(* Logix 5000 project; controller STAT 1756-L72 rev 20.12; software revision 20.04; part 19 of 34 *)
(* tags used below, declared in another part *)
   B14 : DINT[30];
   B16 : DINT[30];
   B17 : DINT[30];
   B3 : DINT[256];
   B9 : DINT[40];
   F8 : REAL[256];
   I1_005_Bit15 : ALIAS FOR I1[5].15;
   I6_000_Bit02 : ALIAS FOR I6[0].2;   // totaal 3 debiet stfa 3
   I6_000_Bit10 : ALIAS FOR I6[0].10;   // pressostaat osmose1
   I6_000_Bit11 : ALIAS FOR I6[0].11;   // pressostaat osmose2
   I6_000_Bit12 : ALIAS FOR I6[0].12;   // pressostaat osmose3
   I6_001_Bit07 : ALIAS FOR I6[1].7;   // pulse debietmeter zandfilter osmose
   N12 : DINT[230];
   N13 : DINT[230];
   N26 : DINT[256];
   O14_000_Bit14 : ALIAS FOR O14[0].14;   // STFA3_EV1 STFA3_EV1
   O14_000_Bit15 : ALIAS FOR O14[0].15;   // STFA3_EV2 STFA3_EV2
   O14_001_Bit00 : ALIAS FOR O14[1].0;   // STFA3_EV3 STFA3_EV3
   O14_001_Bit01 : ALIAS FOR O14[1].1;   // STFA3_EV4 STFA3_EV4
   O14_001_Bit02 : ALIAS FOR O14[1].2;   // STFA3_EV5 STFA3_EV5
   O14_001_Bit03 : ALIAS FOR O14[1].3;   // STFA3_EV6 STFA3_EV6
   O14_001_Bit12 : ALIAS FOR O14[1].12;   // RO1_EV1 RO1_EV1
   O14_001_Bit13 : ALIAS FOR O14[1].13;   // RO1_EV2 RO1_EV2
   O15_000_Bit00 : ALIAS FOR O15[0].0;   // RO2_EV1 RO2_EV1
   O15_000_Bit01 : ALIAS FOR O15[0].1;   // RO2_EV2 RO2_EV2
   T27 : TIMER[100];
   T4 : TIMER[200];
(* ibt, continued *)

ROUTINE _22_SEQ_VERZ3   (* ladder *)
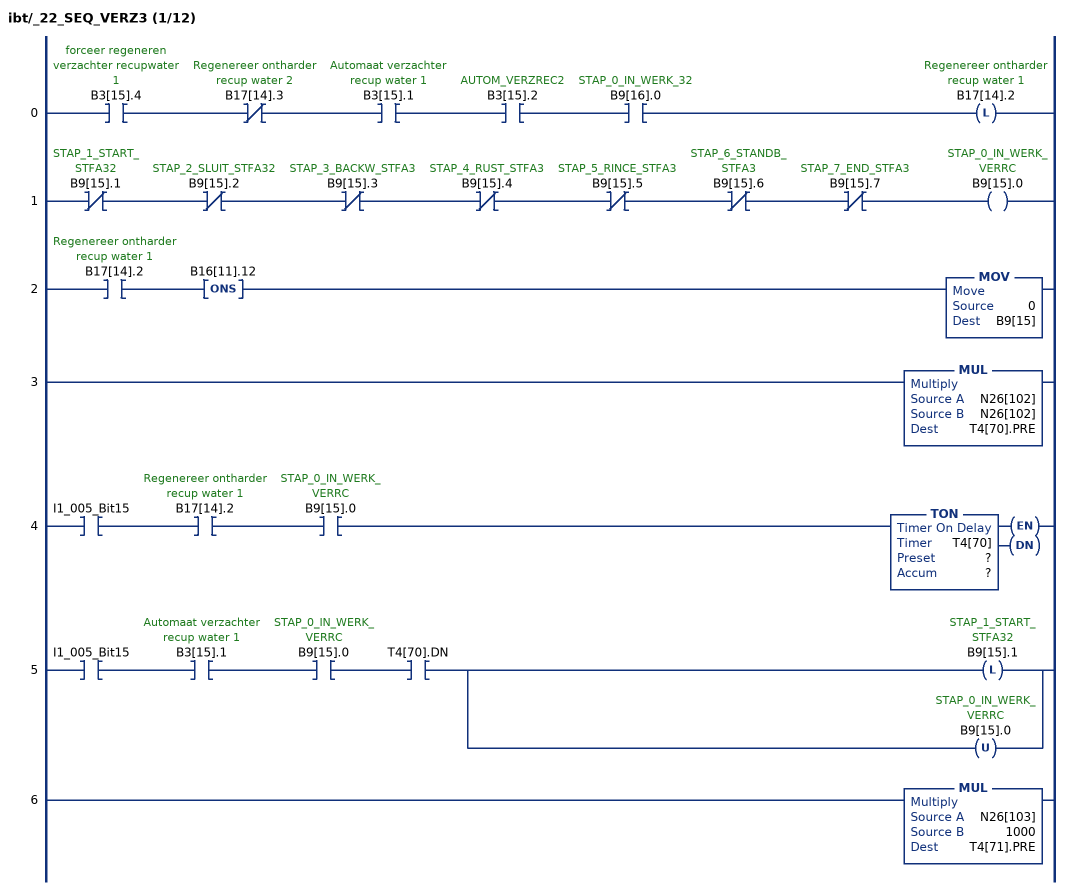
   0: XIC(B3[15].4)XIO(B17[14].3)XIC(B3[15].1)XIC(B3[15].2)XIC(B9[16].0)OTL(B17[14].2);
   1: XIO(B9[15].1)XIO(B9[15].2)XIO(B9[15].3)XIO(B9[15].4)XIO(B9[15].5)XIO(B9[15].6)XIO(B9[15].7)OTE(B9[15].0);
   2: XIC(B17[14].2)ONS(B16[11].12)MOV(0,B9[15]);
   3: MUL(N26[102],N26[102],T4[70].PRE);
   4: XIC(I1_005_Bit15)XIC(B17[14].2)XIC(B9[15].0)TON(T4[70],?,?);
   5: XIC(I1_005_Bit15)XIC(B3[15].1)XIC(B9[15].0)XIC(T4[70].DN)[OTL(B9[15].1) ,OTU(B9[15].0) ];
   6: MUL(N26[103],1000,T4[71].PRE);
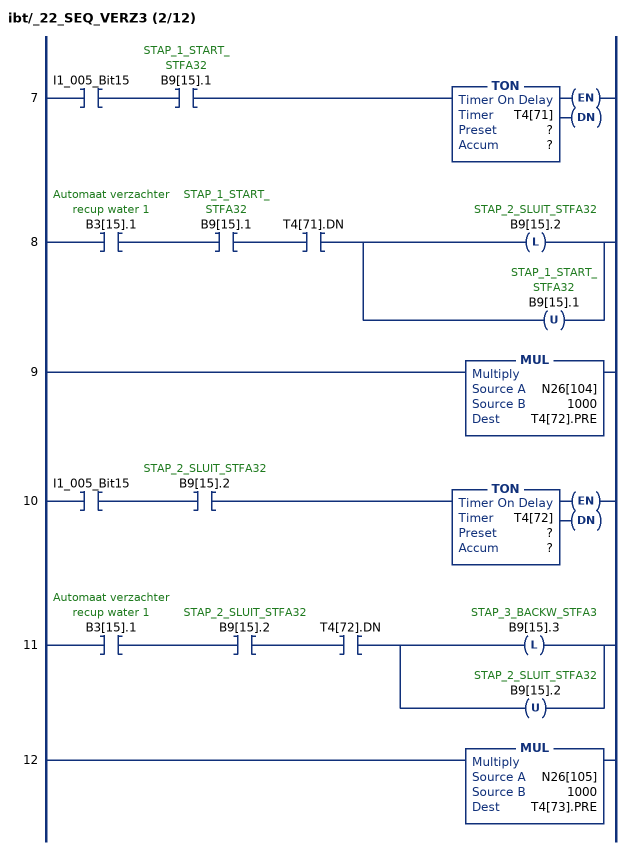
   7: XIC(I1_005_Bit15)XIC(B9[15].1)TON(T4[71],?,?);
   8: XIC(B3[15].1)XIC(B9[15].1)XIC(T4[71].DN)[OTL(B9[15].2) ,OTU(B9[15].1) ];
   9: MUL(N26[104],1000,T4[72].PRE);
   10: XIC(I1_005_Bit15)XIC(B9[15].2)TON(T4[72],?,?);
   11: XIC(B3[15].1)XIC(B9[15].2)XIC(T4[72].DN)[OTL(B9[15].3) ,OTU(B9[15].2) ];
   12: MUL(N26[105],1000,T4[73].PRE);
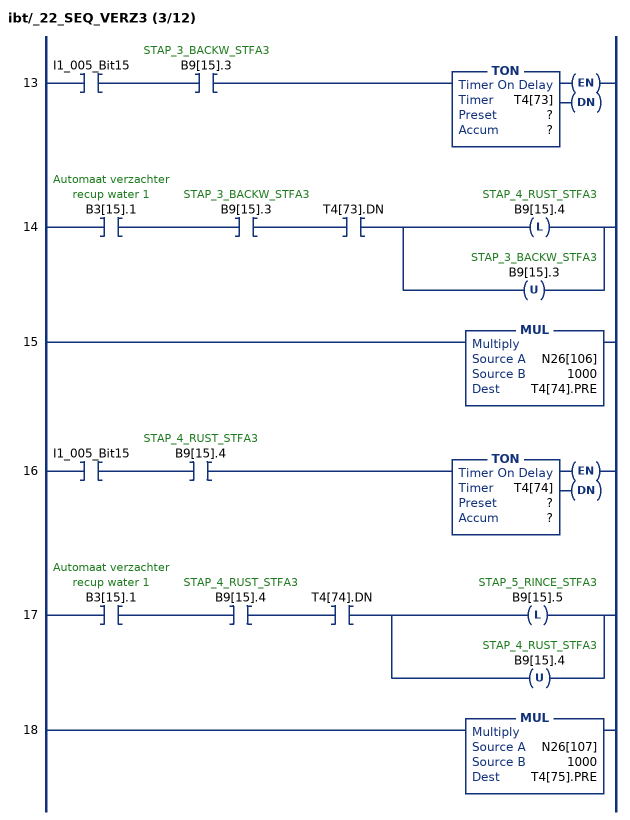
   13: XIC(I1_005_Bit15)XIC(B9[15].3)TON(T4[73],?,?);
   14: XIC(B3[15].1)XIC(B9[15].3)XIC(T4[73].DN)[OTL(B9[15].4) ,OTU(B9[15].3) ];
   15: MUL(N26[106],1000,T4[74].PRE);
   16: XIC(I1_005_Bit15)XIC(B9[15].4)TON(T4[74],?,?);
   17: XIC(B3[15].1)XIC(B9[15].4)XIC(T4[74].DN)[OTL(B9[15].5) ,OTU(B9[15].4) ];
   18: MUL(N26[107],1000,T4[75].PRE);
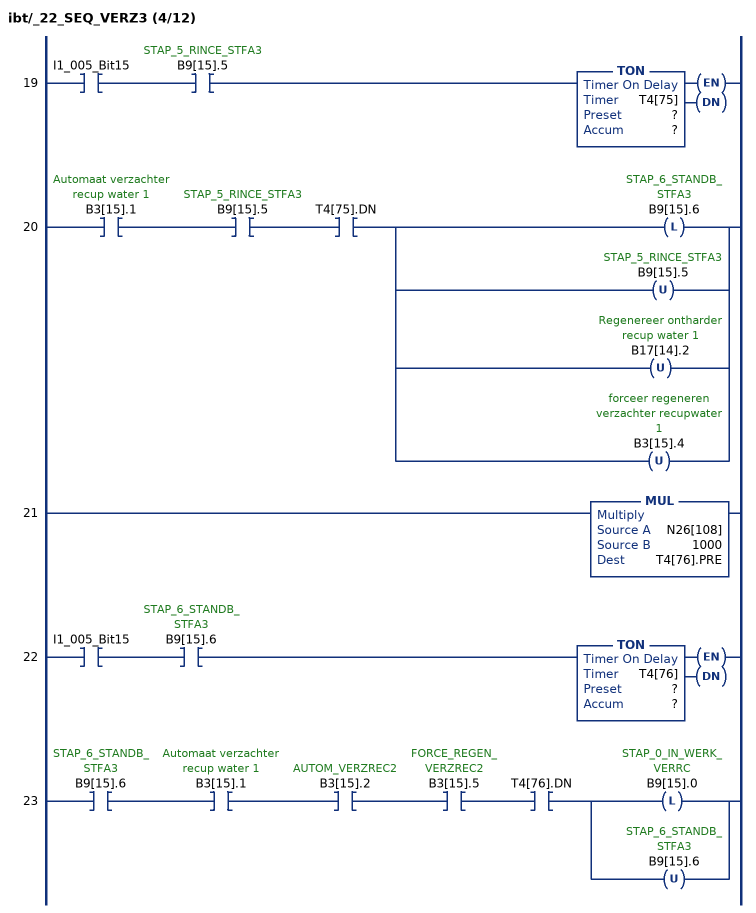
   19: XIC(I1_005_Bit15)XIC(B9[15].5)TON(T4[75],?,?);
   20: XIC(B3[15].1)XIC(B9[15].5)XIC(T4[75].DN)[OTL(B9[15].6) ,[OTU(B9[15].5) ,[OTU(B17[14].2) ,OTU(B3[15].4) ] ] ];
   21: MUL(N26[108],1000,T4[76].PRE);
   22: XIC(I1_005_Bit15)XIC(B9[15].6)TON(T4[76],?,?);
   23: XIC(B9[15].6)XIC(B3[15].1)XIC(B3[15].2)XIC(B3[15].5)XIC(T4[76].DN)[OTL(B9[15].0) ,OTU(B9[15].6) ];
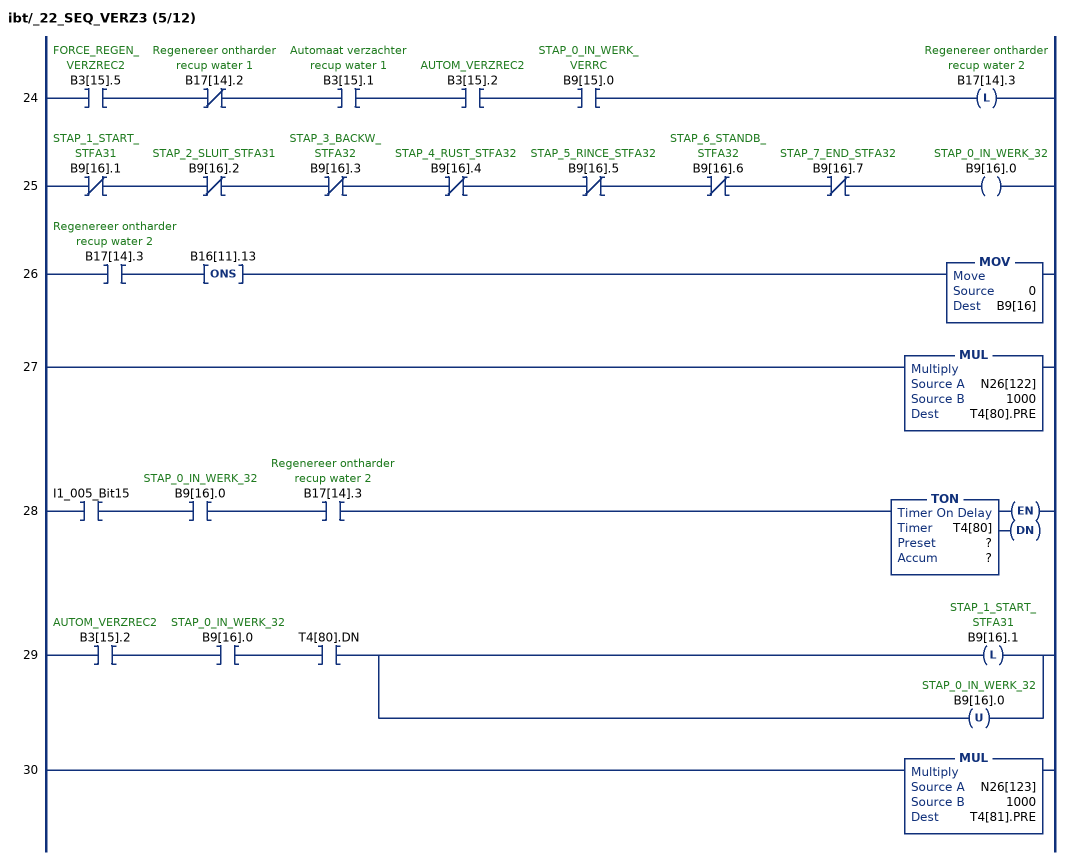
   24: XIC(B3[15].5)XIO(B17[14].2)XIC(B3[15].1)XIC(B3[15].2)XIC(B9[15].0)OTL(B17[14].3);
   25: XIO(B9[16].1)XIO(B9[16].2)XIO(B9[16].3)XIO(B9[16].4)XIO(B9[16].5)XIO(B9[16].6)XIO(B9[16].7)OTE(B9[16].0);
   26: XIC(B17[14].3)ONS(B16[11].13)MOV(0,B9[16]);
   27: MUL(N26[122],1000,T4[80].PRE);
   28: XIC(I1_005_Bit15)XIC(B9[16].0)XIC(B17[14].3)TON(T4[80],?,?);
   29: XIC(B3[15].2)XIC(B9[16].0)XIC(T4[80].DN)[OTL(B9[16].1) ,OTU(B9[16].0) ];
   30: MUL(N26[123],1000,T4[81].PRE);
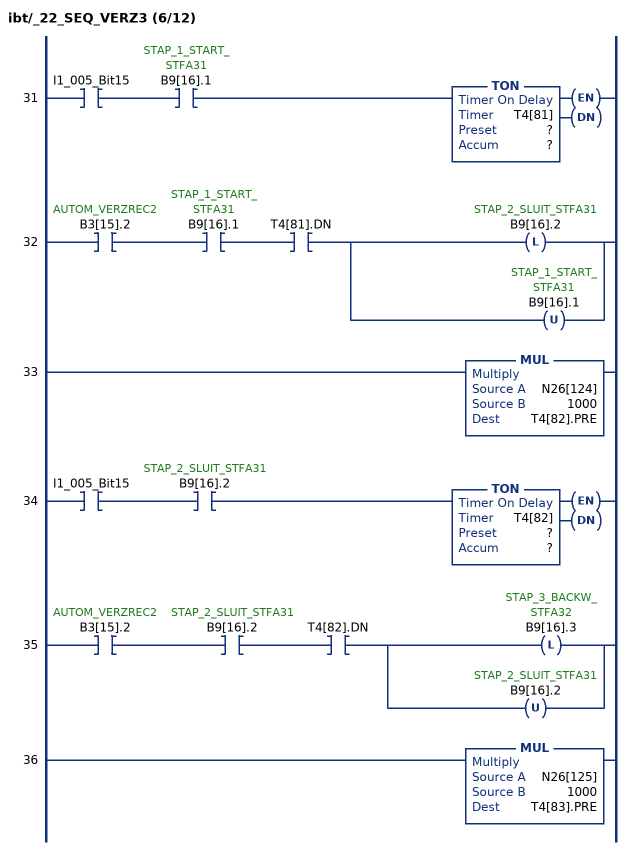
   31: XIC(I1_005_Bit15)XIC(B9[16].1)TON(T4[81],?,?);
   32: XIC(B3[15].2)XIC(B9[16].1)XIC(T4[81].DN)[OTL(B9[16].2) ,OTU(B9[16].1) ];
   33: MUL(N26[124],1000,T4[82].PRE);
   34: XIC(I1_005_Bit15)XIC(B9[16].2)TON(T4[82],?,?);
   35: XIC(B3[15].2)XIC(B9[16].2)XIC(T4[82].DN)[OTL(B9[16].3) ,OTU(B9[16].2) ];
   36: MUL(N26[125],1000,T4[83].PRE);
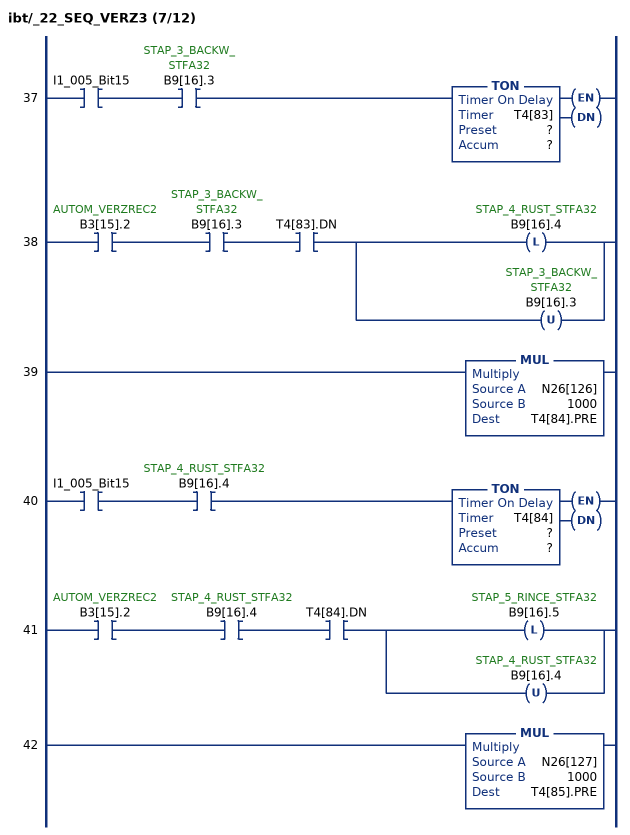
   37: XIC(I1_005_Bit15)XIC(B9[16].3)TON(T4[83],?,?);
   38: XIC(B3[15].2)XIC(B9[16].3)XIC(T4[83].DN)[OTL(B9[16].4) ,OTU(B9[16].3) ];
   39: MUL(N26[126],1000,T4[84].PRE);
   40: XIC(I1_005_Bit15)XIC(B9[16].4)TON(T4[84],?,?);
   41: XIC(B3[15].2)XIC(B9[16].4)XIC(T4[84].DN)[OTL(B9[16].5) ,OTU(B9[16].4) ];
   42: MUL(N26[127],1000,T4[85].PRE);
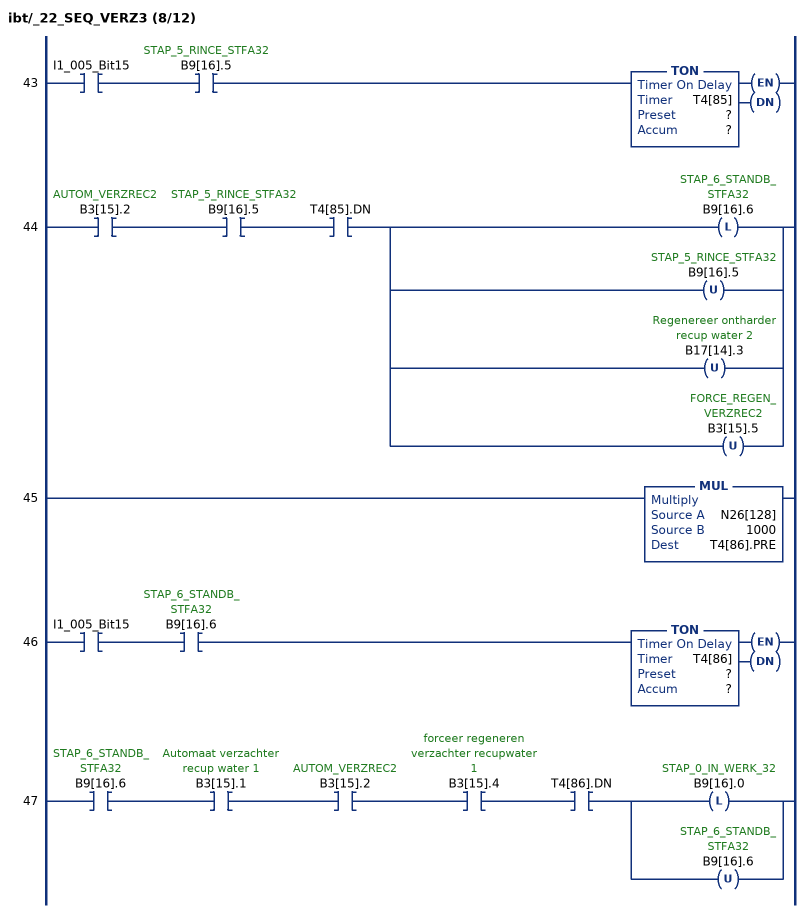
   43: XIC(I1_005_Bit15)XIC(B9[16].5)TON(T4[85],?,?);
   44: XIC(B3[15].2)XIC(B9[16].5)XIC(T4[85].DN)[OTL(B9[16].6) ,[OTU(B9[16].5) ,[OTU(B17[14].3) ,OTU(B3[15].5) ] ] ];
   45: MUL(N26[128],1000,T4[86].PRE);
   46: XIC(I1_005_Bit15)XIC(B9[16].6)TON(T4[86],?,?);
   47: XIC(B9[16].6)XIC(B3[15].1)XIC(B3[15].2)XIC(B3[15].4)XIC(T4[86].DN)[OTL(B9[16].0) ,OTU(B9[16].6) ];
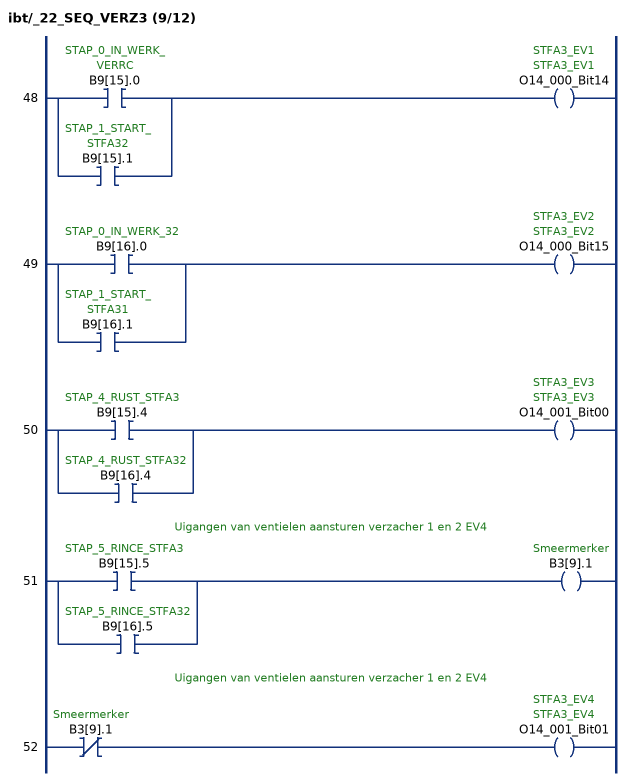
   48: [XIC(B9[15].0) ,XIC(B9[15].1) ]OTE(O14_000_Bit14);
   49: [XIC(B9[16].0) ,XIC(B9[16].1) ]OTE(O14_000_Bit15);
   50: [XIC(B9[15].4) ,XIC(B9[16].4) ]OTE(O14_001_Bit00);
   // Uigangen van ventielen aansturen verzacher 1 en 2 EV4
   51: [XIC(B9[15].5) ,XIC(B9[16].5) ]OTE(B3[9].1);
   // Uigangen van ventielen aansturen verzacher 1 en 2 EV4
   52: XIO(B3[9].1)OTE(O14_001_Bit01);
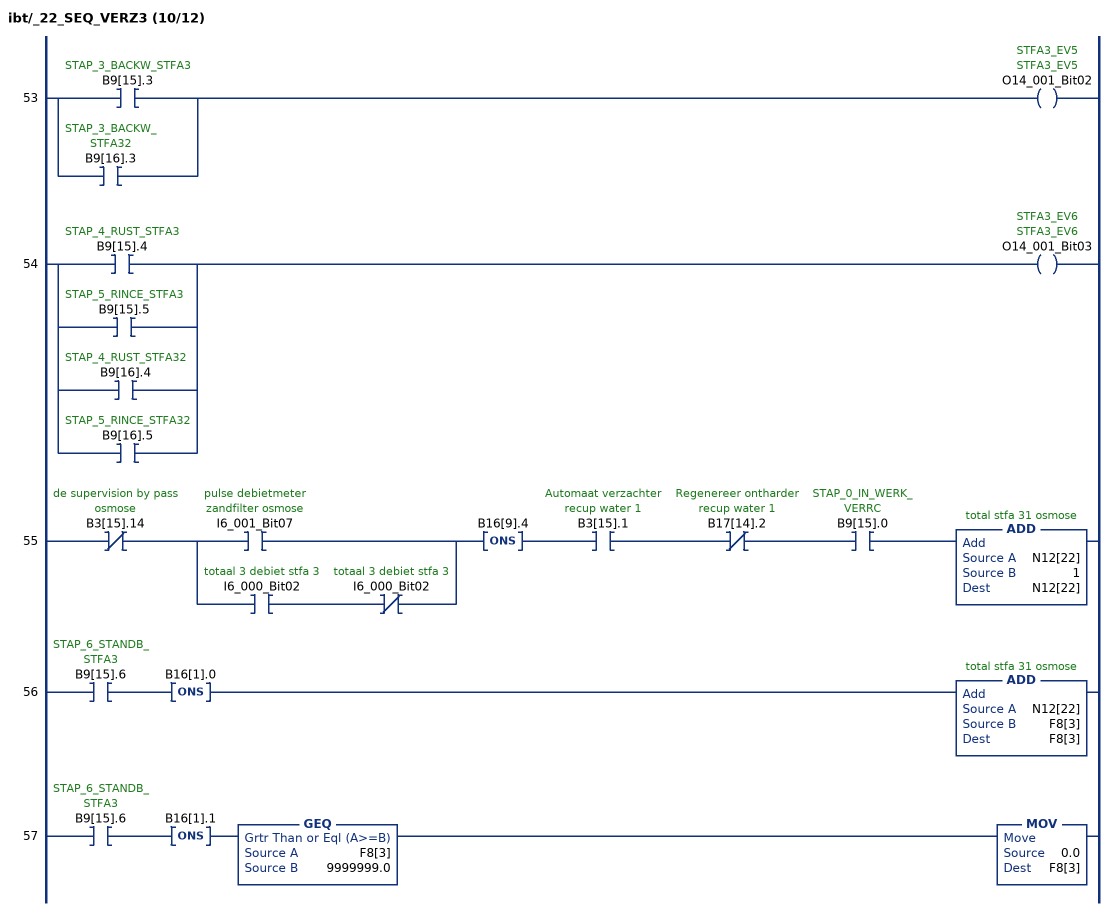
   53: [XIC(B9[15].3) ,XIC(B9[16].3) ]OTE(O14_001_Bit02);
   54: [XIC(B9[15].4) ,[XIC(B9[15].5) ,[XIC(B9[16].4) ,XIC(B9[16].5) ] ] ]OTE(O14_001_Bit03);
   55: XIO(B3[15].14)[XIC(I6_001_Bit07) ,XIC(I6_000_Bit02) XIO(I6_000_Bit02) ]ONS(B16[9].4)XIC(B3[15].1)XIO(B17[14].2)XIC(B9[15].0)ADD(N12[22],1,N12[22]);
   56: XIC(B9[15].6)ONS(B16[1].0)ADD(N12[22],F8[3],F8[3]);
   57: XIC(B9[15].6)ONS(B16[1].1)GEQ(F8[3],9999999.0)MOV(0.0,F8[3]);
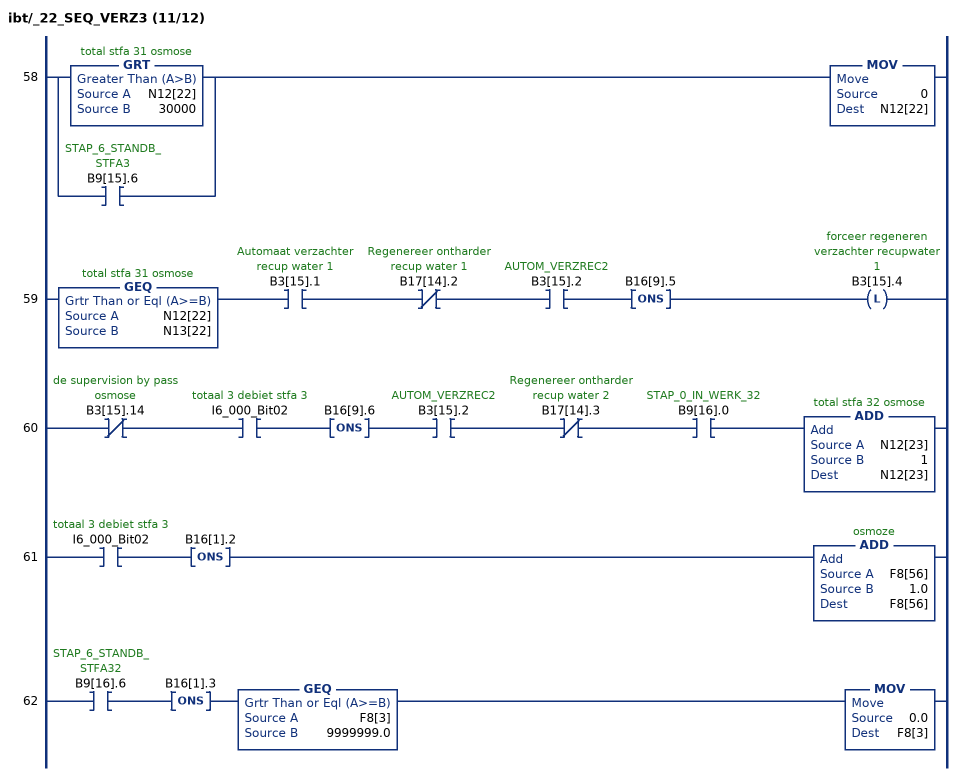
   58: [GRT(N12[22],30000) ,XIC(B9[15].6) ]MOV(0,N12[22]);
   59: GEQ(N12[22],N13[22])XIC(B3[15].1)XIO(B17[14].2)XIC(B3[15].2)ONS(B16[9].5)OTL(B3[15].4);
   60: XIO(B3[15].14)XIC(I6_000_Bit02)ONS(B16[9].6)XIC(B3[15].2)XIO(B17[14].3)XIC(B9[16].0)ADD(N12[23],1,N12[23]);
   61: XIC(I6_000_Bit02)ONS(B16[1].2)ADD(F8[56],1.0,F8[56]);
   62: XIC(B9[16].6)ONS(B16[1].3)GEQ(F8[3],9999999.0)MOV(0.0,F8[3]);
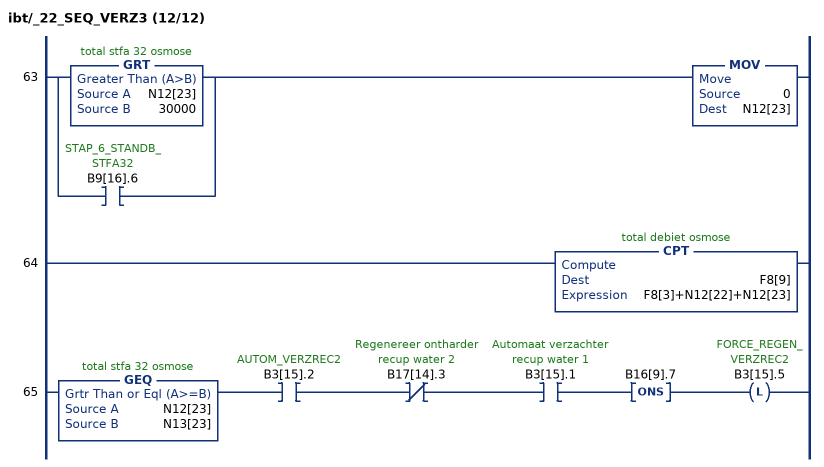
   63: [GRT(N12[23],30000) ,XIC(B9[16].6) ]MOV(0,N12[23]);
   64: CPT(F8[9],F8[3]+N12[22]+N12[23]);
   65: GEQ(N12[23],N13[23])XIC(B3[15].2)XIO(B17[14].3)XIC(B3[15].1)ONS(B16[9].7)OTL(B3[15].5);
END_ROUTINE

ROUTINE _23_SEQ_OSMOSE   (* ladder *)
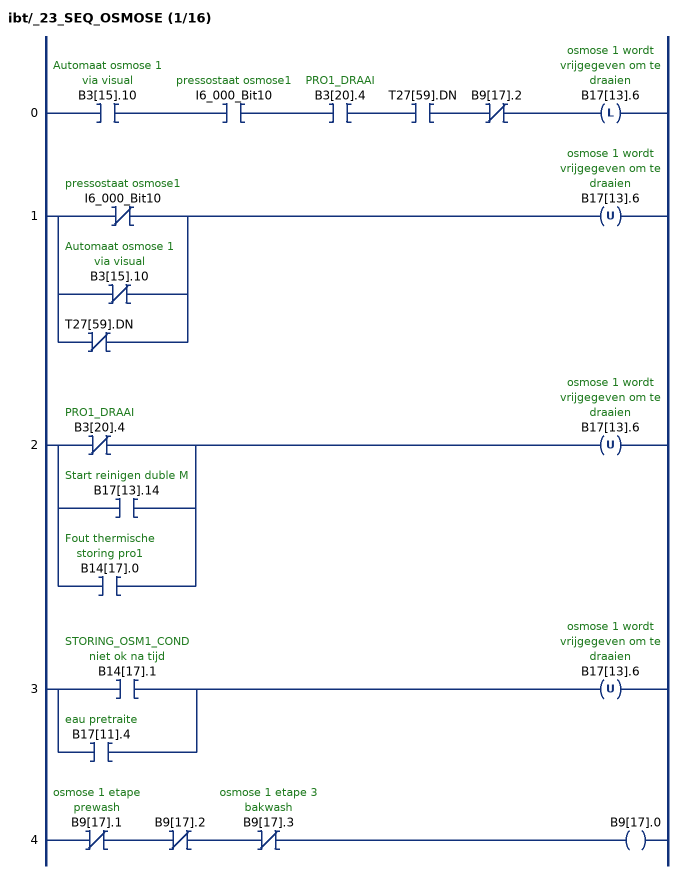
   0: XIC(B3[15].10)XIC(I6_000_Bit10)XIC(B3[20].4)XIC(T27[59].DN)XIO(B9[17].2)OTL(B17[13].6);
   1: [XIO(I6_000_Bit10) ,[XIO(B3[15].10) ,XIO(T27[59].DN) ] ]OTU(B17[13].6);
   2: [XIO(B3[20].4) ,[XIC(B17[13].14) ,XIC(B14[17].0) ] ]OTU(B17[13].6);
   3: [XIC(B14[17].1) ,XIC(B17[11].4) ]OTU(B17[13].6);
   4: XIO(B9[17].1)XIO(B9[17].2)XIO(B9[17].3)OTE(B9[17].0);
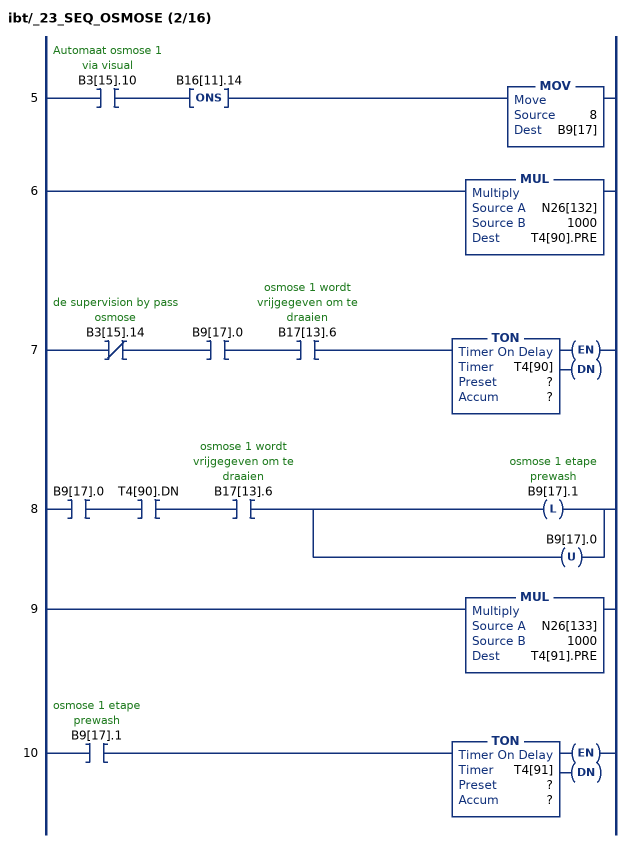
   5: XIC(B3[15].10)ONS(B16[11].14)MOV(8,B9[17]);
   6: MUL(N26[132],1000,T4[90].PRE);
   7: XIO(B3[15].14)XIC(B9[17].0)XIC(B17[13].6)TON(T4[90],?,?);
   8: XIC(B9[17].0)XIC(T4[90].DN)XIC(B17[13].6)[OTL(B9[17].1) ,OTU(B9[17].0) ];
   9: MUL(N26[133],1000,T4[91].PRE);
   10: XIC(B9[17].1)TON(T4[91],?,?);
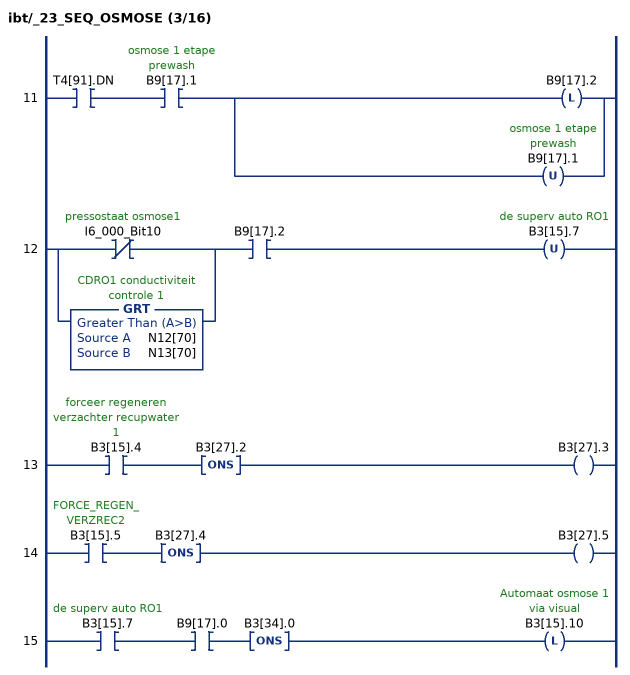
   11: XIC(T4[91].DN)XIC(B9[17].1)[OTL(B9[17].2) ,OTU(B9[17].1) ];
   12: [XIO(I6_000_Bit10) ,GRT(N12[70],N13[70]) ]XIC(B9[17].2)OTU(B3[15].7);
   13: XIC(B3[15].4)ONS(B3[27].2)OTE(B3[27].3);
   14: XIC(B3[15].5)ONS(B3[27].4)OTE(B3[27].5);
   15: XIC(B3[15].7)XIC(B9[17].0)ONS(B3[34].0)OTL(B3[15].10);
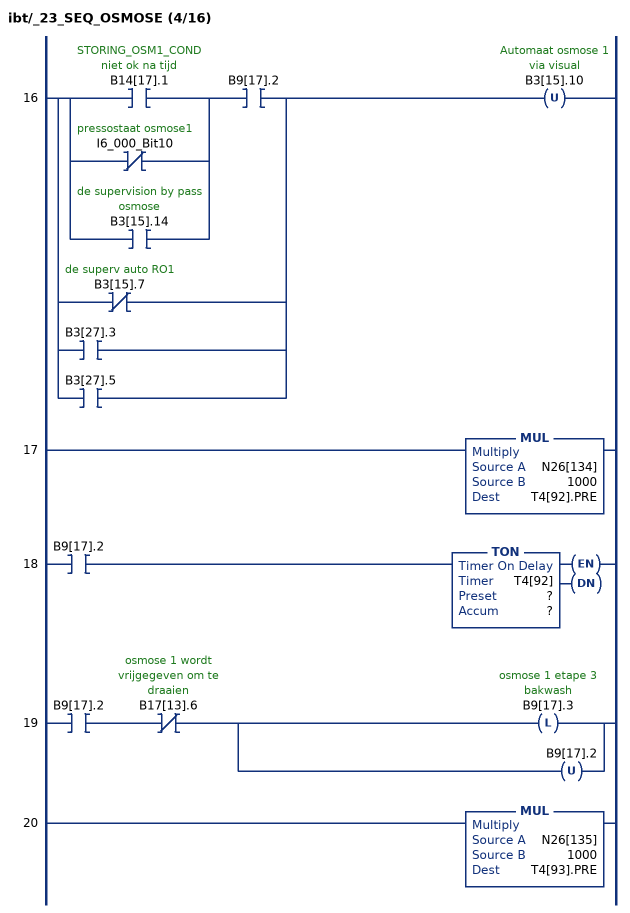
   16: [[XIC(B14[17].1) ,[XIO(I6_000_Bit10) ,XIC(B3[15].14) ] ] XIC(B9[17].2) ,XIO(B3[15].7) ,XIC(B3[27].3) ,XIC(B3[27].5) ]OTU(B3[15].10);
   17: MUL(N26[134],1000,T4[92].PRE);
   18: XIC(B9[17].2)TON(T4[92],?,?);
   19: XIC(B9[17].2)XIO(B17[13].6)[OTL(B9[17].3) ,OTU(B9[17].2) ];
   20: MUL(N26[135],1000,T4[93].PRE);
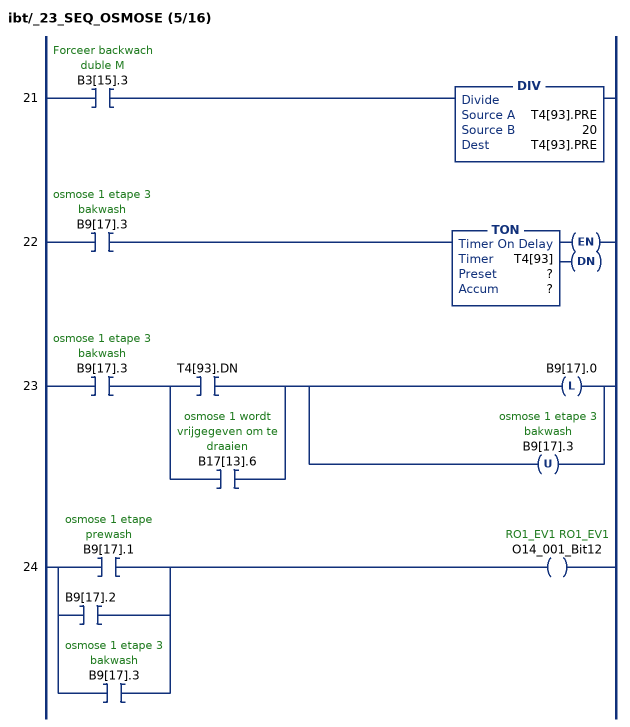
   21: XIC(B3[15].3)DIV(T4[93].PRE,20,T4[93].PRE);
   22: XIC(B9[17].3)TON(T4[93],?,?);
   23: XIC(B9[17].3)[XIC(T4[93].DN) ,XIC(B17[13].6) ][OTL(B9[17].0) ,OTU(B9[17].3) ];
   24: [XIC(B9[17].1) ,[XIC(B9[17].2) ,XIC(B9[17].3) ] ]OTE(O14_001_Bit12);
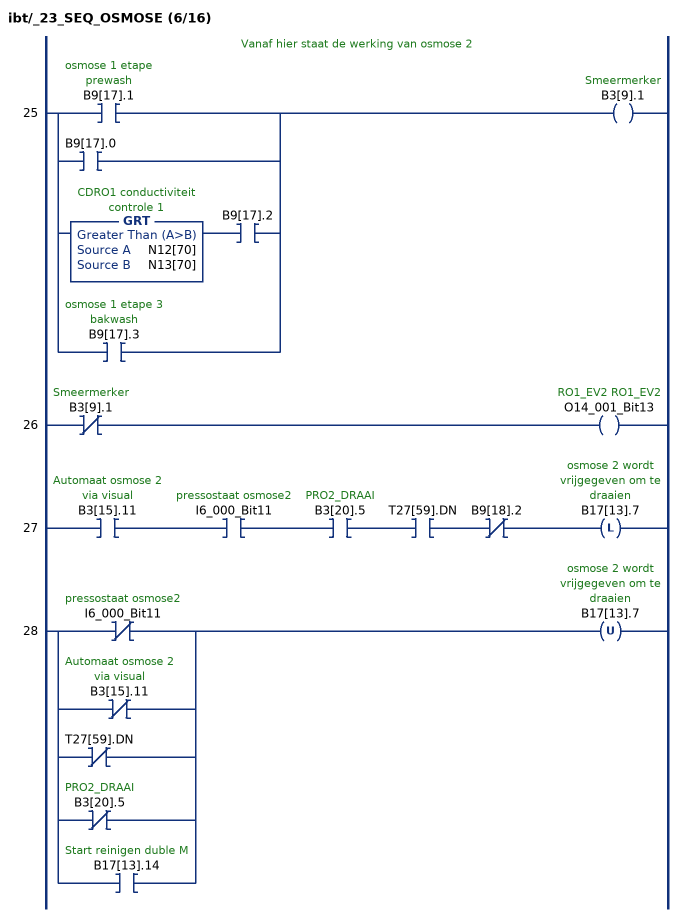
   // Vanaf hier staat de werking van osmose 2
   25: [[XIC(B9[17].1) ,XIC(B9[17].0) ] ,[GRT(N12[70],N13[70]) XIC(B9[17].2) ,XIC(B9[17].3) ] ]OTE(B3[9].1);
   26: XIO(B3[9].1)OTE(O14_001_Bit13);
   27: XIC(B3[15].11)XIC(I6_000_Bit11)XIC(B3[20].5)XIC(T27[59].DN)XIO(B9[18].2)OTL(B17[13].7);
   28: [XIO(I6_000_Bit11) ,[XIO(B3[15].11) ,[[XIO(T27[59].DN) ,XIO(B3[20].5) ] ,XIC(B17[13].14) ] ] ]OTU(B17[13].7);
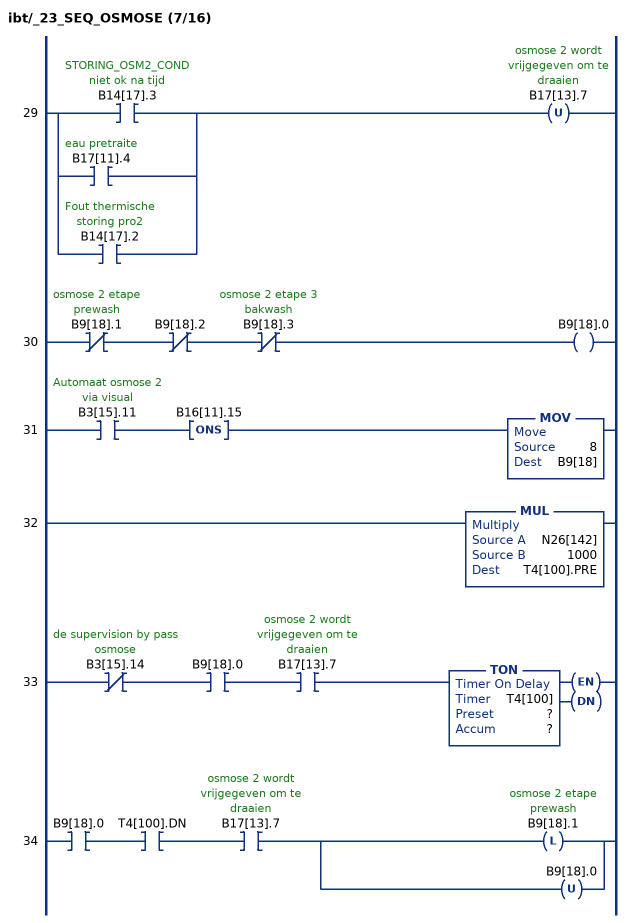
   29: [XIC(B14[17].3) ,[XIC(B17[11].4) ,XIC(B14[17].2) ] ]OTU(B17[13].7);
   30: XIO(B9[18].1)XIO(B9[18].2)XIO(B9[18].3)OTE(B9[18].0);
   31: XIC(B3[15].11)ONS(B16[11].15)MOV(8,B9[18]);
   32: MUL(N26[142],1000,T4[100].PRE);
   33: XIO(B3[15].14)XIC(B9[18].0)XIC(B17[13].7)TON(T4[100],?,?);
   34: XIC(B9[18].0)XIC(T4[100].DN)XIC(B17[13].7)[OTL(B9[18].1) ,OTU(B9[18].0) ];
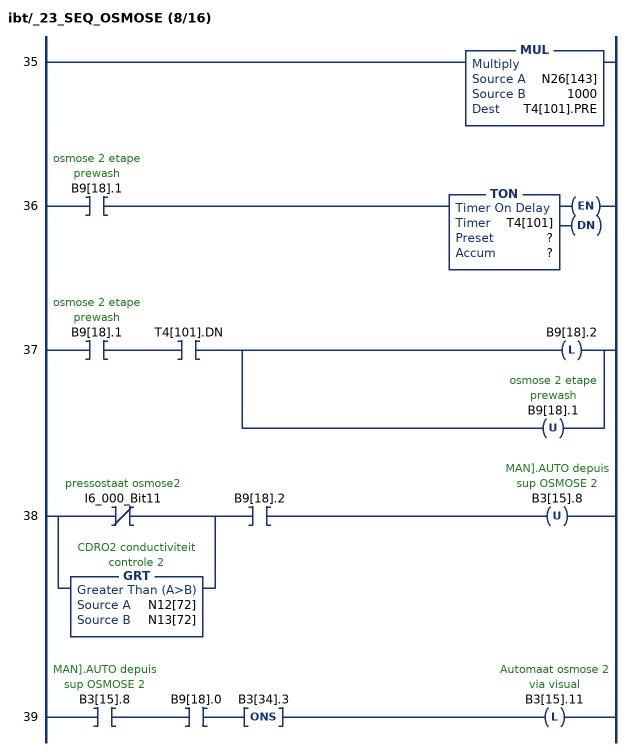
   35: MUL(N26[143],1000,T4[101].PRE);
   36: XIC(B9[18].1)TON(T4[101],?,?);
   37: XIC(B9[18].1)XIC(T4[101].DN)[OTL(B9[18].2) ,OTU(B9[18].1) ];
   38: [XIO(I6_000_Bit11) ,GRT(N12[72],N13[72]) ]XIC(B9[18].2)OTU(B3[15].8);
   39: XIC(B3[15].8)XIC(B9[18].0)ONS(B3[34].3)OTL(B3[15].11);
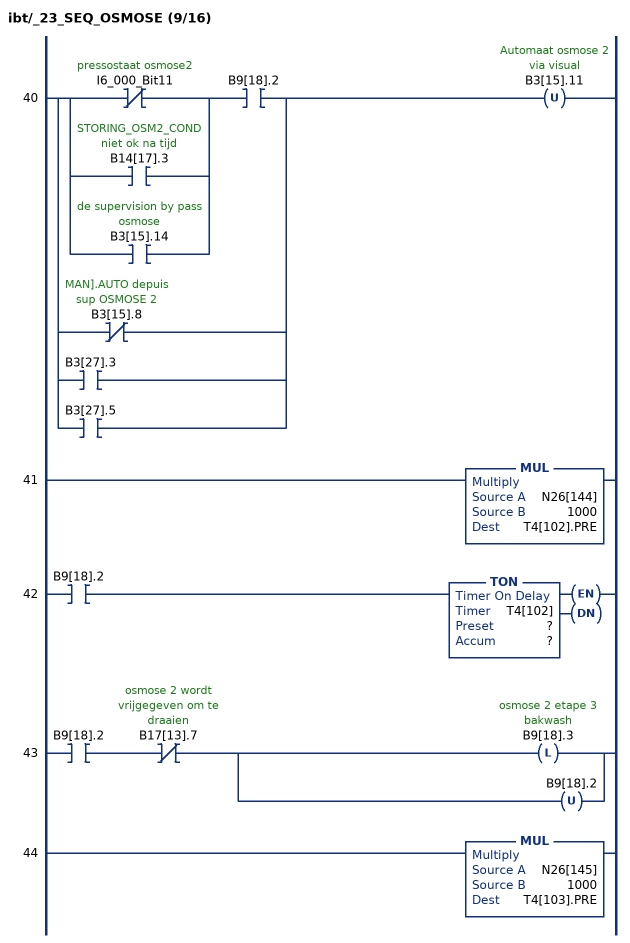
   40: [[XIO(I6_000_Bit11) ,XIC(B14[17].3) ,XIC(B3[15].14) ] XIC(B9[18].2) ,XIO(B3[15].8) ,XIC(B3[27].3) ,XIC(B3[27].5) ]OTU(B3[15].11);
   41: MUL(N26[144],1000,T4[102].PRE);
   42: XIC(B9[18].2)TON(T4[102],?,?);
   43: XIC(B9[18].2)XIO(B17[13].7)[OTL(B9[18].3) ,OTU(B9[18].2) ];
   44: MUL(N26[145],1000,T4[103].PRE);
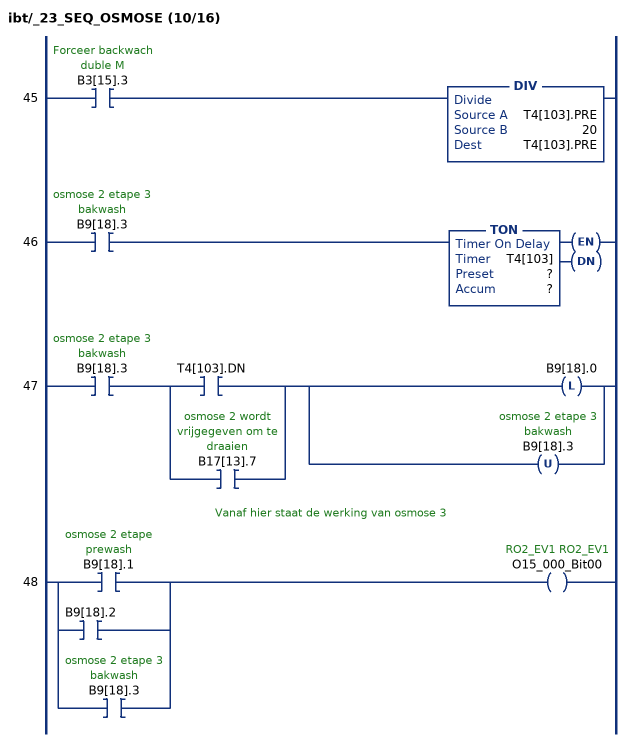
   45: XIC(B3[15].3)DIV(T4[103].PRE,20,T4[103].PRE);
   46: XIC(B9[18].3)TON(T4[103],?,?);
   47: XIC(B9[18].3)[XIC(T4[103].DN) ,XIC(B17[13].7) ][OTL(B9[18].0) ,OTU(B9[18].3) ];
   // Vanaf hier staat de werking van osmose 3
   48: [XIC(B9[18].1) ,[XIC(B9[18].2) ,XIC(B9[18].3) ] ]OTE(O15_000_Bit00);
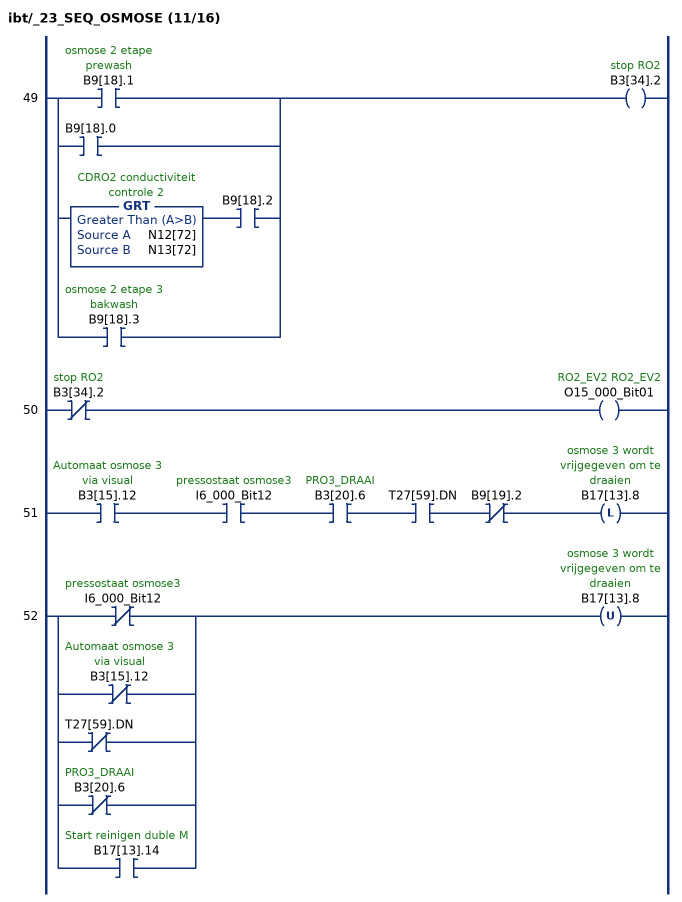
   49: [[XIC(B9[18].1) ,XIC(B9[18].0) ] ,[GRT(N12[72],N13[72]) XIC(B9[18].2) ,XIC(B9[18].3) ] ]OTE(B3[34].2);
   50: XIO(B3[34].2)OTE(O15_000_Bit01);
   51: XIC(B3[15].12)XIC(I6_000_Bit12)XIC(B3[20].6)XIC(T27[59].DN)XIO(B9[19].2)OTL(B17[13].8);
   52: [XIO(I6_000_Bit12) ,[XIO(B3[15].12) ,[XIO(T27[59].DN) ,[XIO(B3[20].6) ,XIC(B17[13].14) ] ] ] ]OTU(B17[13].8);
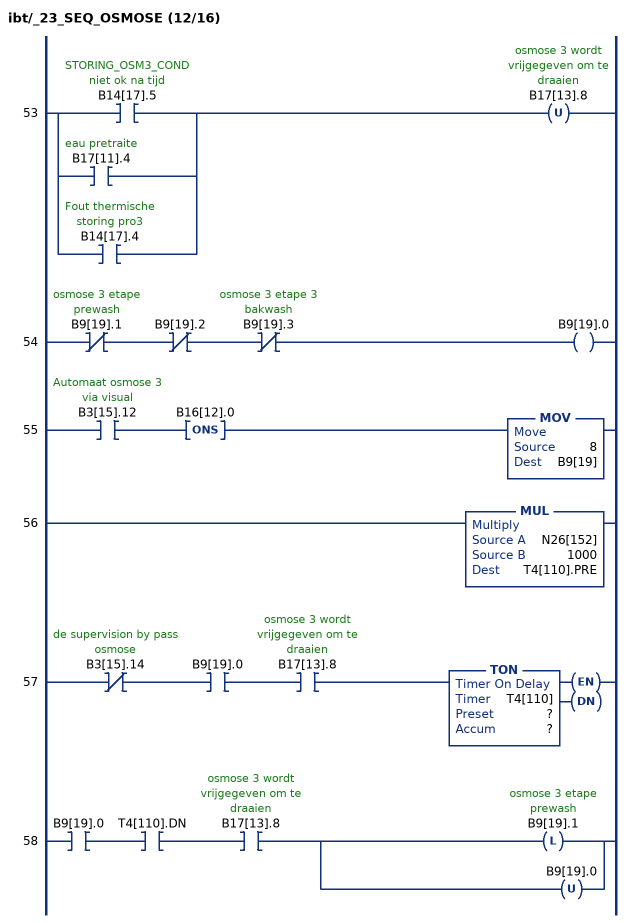
   53: [XIC(B14[17].5) ,[XIC(B17[11].4) ,XIC(B14[17].4) ] ]OTU(B17[13].8);
   54: XIO(B9[19].1)XIO(B9[19].2)XIO(B9[19].3)OTE(B9[19].0);
   55: XIC(B3[15].12)ONS(B16[12].0)MOV(8,B9[19]);
   56: MUL(N26[152],1000,T4[110].PRE);
   57: XIO(B3[15].14)XIC(B9[19].0)XIC(B17[13].8)TON(T4[110],?,?);
   58: XIC(B9[19].0)XIC(T4[110].DN)XIC(B17[13].8)[OTL(B9[19].1) ,OTU(B9[19].0) ];
